{attribute 'pack_mode' := '1'} 
TYPE ASCF_CC_OPCUACS_Reader_Temp_String :
STRUCT
	stReadListReturnInfo	: ARRAY [1..2] OF ST_UAReadListReturnInfo;
	QC		: BYTE		:= 16#0;
	Value	: STRING	:= '';
END_STRUCT
END_TYPE

(* stored: Version 1.1.0.1, ProductVersion 3.1.4026.4
   DUT ASCF_CC_OPCUACS_Reader_Temp_String: Id {63b2bac8-b490-487f-b1b7-f58be1d16136} *)
